// TIA Portal V19 export
DATA_BLOCK "Config"   // DB51
// stored: MemoryReserve 100, Namespace Unit.Em1
   VAR
      em { ExternalWritable := 'False'} : "LAF_typeEmConfiguration";   // Configuration of EM Parameters
   END_VAR
BEGIN
   em.referenceDesignator.parent := WSTRING#'Unit';
   em.referenceDesignator.relative := WSTRING#'EM1';
END_DATA_BLOCK
